# EPICS autosave request: iocs/aravisIOC/iocBoot/iocAravis/auto_settings.req
file "aravisCamera_settings.req", P=$(P),  R=cam1:
file "NDStdArrays_settings.req",  P=$(P),  R=image1:
file "commonPlugin_settings.req", P=$(P)

$(P)cam1:GC_Gamma
$(P)cam1:GC_GevSCPSPacketSize
